FUNCTION_BLOCK TcoFeedingSequenceTask EXTENDS TcoCore.TcoTask
VAR
	_sequence      : TcoCore.TcoSequence(THIS^, eRestoreMode.None);
    _observerSequence       : TcoCore.TcoSequencerObserver(THIS^);
END_VAR

PROPERTY PUBLIC Observer : REFERENCE TO TcoCore.TcoSequencerObserver
GET
Observer ref=_observerSequence;
END_GET
END_PROPERTY

(*~
	<docu>
		<summary>
			Restores this instance to the Ready state. Can be called explicitly or from within one of the restore mechanisms.
			<para>
				See also <see cref="PlcDocu.TcoCore.TcoTask.AutoRestorable()"/>
			</para>
		</summary>			
	</docu>	
~*)
METHOD Restore : ITcoRestorable
SUPER^.Restore();
_sequence.Restore();
END_METHOD

PROPERTY PUBLIC Sequence : REFERENCE TO TcoCore.TcoSequence
GET
Sequence ref=_sequence;
END_GET
END_PROPERTY

END_FUNCTION_BLOCK

(* stored: Version 1.1.0.1
   POU TcoFeedingSequenceTask: Id {6a15bf14-7b1b-4cbd-8547-7cf38af9c488}, SpecialFunc None
   Property Observer: Id {9113932a-5f79-4cb8-913e-f1f163042dcd}
   Get Get: Id {2c81941f-30e5-4583-aacb-87ec3829c12b}
   Method Restore: Id {70622ba5-65b1-4df5-a40b-3f44610a5cf5}
   Property Sequence: Id {94bbc59b-0664-426f-bfe4-95dc7aefb9fd}
   Get Get: Id {ac4daf50-fcf1-445e-abd1-05fe37c35ab0} *)
